(* PLC project apnew, Dassault Systèmes ControlBuild 2024x Refresh1 *)
(* stored: creationDateTime 2024-04-12T14:40:36-01:00 *)

PROGRAM apnew.apnew

(* FBD diagram, written out as Structured Text *)
END_PROGRAM
